// TwinCAT 3 PLC project Samples
// Title: TF8040 PLC-Samples
// Company: Beckhoff Automation GmbH
// Author: Beckhoff Automation
// ProjectVersion: 2.1.2.0
// Description: PLC.Samples to demontrate function volume of TF8040.
// ProgramVersion: 3.1.4026.20
// libraries:
//   Tc2_Standard, * (Beckhoff Automation GmbH)
//   Tc2_System, * (Beckhoff Automation GmbH)
//   Tc2_Utilities, * (Beckhoff Automation GmbH)
//   Tc3_BA2, * (Beckhoff Automation GmbH)
//   Tc3_BA2_Common, * (Beckhoff Automation GmbH)
//   Tc3_BACnetRev14, * (Beckhoff Automation GmbH)
//   Tc3_Module, * (Beckhoff Automation GmbH)
//   Tc3_XBA, * (Beckhoff Automation GmbH)
// project tree:
//   / PlcTask.TcTTO (not stored)
//   SAMPLES/Demo/Event/ FB_Evt_Ack.TcPOU, FB_Evt_EventClasses.TcPOU (not stored), FB_Evt_Events.TcPOU (not stored), FB_Evt_Misc.TcPOU, FB_Evt_QueryCnd.TcPOU
//   SAMPLES/Demo/Event/Function/ F_AcknowledgeEventClass.TcPOU, F_CountEventClassActive.TcPOU
//   SAMPLES/Demo/Objects/ FB_Obj_AddParam.TcPOU (not stored), FB_Obj_General.TcPOU (not stored), FB_Obj_Misc.TcPOU (not stored), FB_Obj_Sequence.TcPOU (not stored), FB_Obj_UserDefined.TcPOU (not stored)
//   SAMPLES/Demo/Objects/Misc/ E_UDef_Mode.TcDUT, FB_UDef_BValEx.TcPOU (not stored), FB_UDef_SpVal.TcPOU (not stored), FB_UDef_SpValEx.TcPOU
//   SAMPLES/Demo/Optional Extensions/Events/ FB_MyLocalObjectEvents.TcPOU, FB_MyProjectEvents.TcPOU
//   SAMPLES/Demo/Optional Extensions/ MAIN_OPTEXT.TcPOU (not stored)
//   SAMPLES/Demo/Other/ FB_Misc.TcPOU (not stored), FB_Texts.TcPOU
//   SAMPLES/Demo/Plant/ FB_Plt_Init1.TcPOU, FB_Plt_Init2.TcPOU, FB_Plt_Init3.TcPOU (not stored)
//   SAMPLES/Demo/Reference/ FB_Ref_Collectors.TcPOU (not stored), FB_Ref_Groups.TcPOU
//   SAMPLES/Demo/Reference/Publish and Subscribe/ FB_Ref_PubSub_Local.TcPOU, FB_Ref_PubSub_Remote.TcPOU (not stored)
//   SAMPLES/Demo/Structure/ FB_Struct_Nested.TcPOU (not stored)
//   SAMPLES/Demo/Supplements/BACnet/ FB_BACnet_EvtInh.TcPOU (not stored), FB_BACnet_ObjPropRef.TcPOU (not stored), FB_BACnet_ObjPropRef_1.TcPOU (not stored), FB_BACnet_RcpList.TcPOU (not stored)
//   SAMPLES/Demo/Supplements/BACnet/Extensions/Events/ FB_BACnet_MyLocalObjectEvents.TcPOU
//   SAMPLES/Demo/Supplements/BACnet/Extensions/ MAIN_OPTEXT_BACnet.TcPOU (not stored)
//   SAMPLES/Demo/[Helper]/FunctionBlocks/Aggregates/ FB_TimerAggregateA.TcPOU (not stored), FB_ProcAggregateB.TcPOU (not stored)
//   SAMPLES/Demo/[Helper]/FunctionBlocks/Nested/ FB_NestedView.TcPOU (not stored), FB_NestedView2.TcPOU (not stored), FB_SubNestedView.TcPOU (not stored), FB_SubSubNestedView.TcPOU (not stored)
//   SAMPLES/ MAIN.TcPOU
//   SAMPLES/Templates/Standard/DUTs/Enumerations/OpMod/ E_OpMod_AC.TcDUT (not stored), E_OpMod_Binary.TcDUT (not stored), E_OpMod_ClsOpn.TcDUT, E_OpMod_Step2.TcDUT
//   SAMPLES/Templates/Standard/GVLs/ MyECIDs.TcGVL, MyLabels.TcGVL (not stored), MyProfiles.TcGVL (not stored)
//   SAMPLES/Templates/Standard/POUs/Trade/General/Building/ FB_BA_Bld01.TcPOU (not stored)
//   SAMPLES/Templates/Standard/POUs/Trade/General/EventClasses/ FB_BA_EC01.TcPOU
//   SAMPLES/Templates/User-defined/Objects/ FB_UDef_Obj.TcPOU
//   SAMPLES/Templates/User-defined/Sample Weather Station/ FB_BA_MyWeatherStation.TcPOU, FB_BA_MyWeatherStationSub.TcPOU, I_BA_MyWeatherStation.TcIO (not stored), ST_BA_MyWeatherData.TcDUT (not stored)
// real-time tasks:
//   TASK PlcTask: cycle T#45ms, priority 20, ADS port 350
//   TASK Device 1 (BACnet IP)_Task_58: cycle T#40ms, priority 58, ADS port 351
//   TASK Gerät 1 (BACnet IP)_QueueTask: cycle T#2ms, priority 8, ADS port 352
// I/O:
//   DEVICE Gerät 1 (BACnet IP), AmsNetId 10.10.1.201.2.1
// variable links:
//   Samples/Samples Instance <-> Device 1 (BACnet IP)
//     PlcTask Inputs/BACnet_Globals.DefaultAdapter.BACnet_AmsNetId <-> Inputs/AmsNetId

// ---- SAMPLES/Demo/Objects/Misc/E_UDef_Mode.TcDUT
{attribute 'qualified_only'}
{attribute 'strict'}

{attribute 'BaParam.Enum.eAdd.DE' := 'Hinzufügen'}
{attribute 'BaParam.Enum.eAdd.EN' := 'Add'}
{attribute 'BaParam.Enum.eSubstract.DE' := 'Abziehen'}
{attribute 'BaParam.Enum.eSubstract.EN' := 'Substract'}
TYPE E_UDef_Mode :
(
	eAdd,
	eSubstract
);
END_TYPE

// ---- SAMPLES/Templates/Standard/DUTs/Enumerations/OpMod/E_OpMod_ClsOpn.TcDUT
{attribute 'qualified_only'}
TYPE E_OpMod_ClsOpn :
(
	eClose			:= 0,
	eOpen			:= 1
	
) UDINT;
END_TYPE

// ---- SAMPLES/Templates/Standard/DUTs/Enumerations/OpMod/E_OpMod_Step2.TcDUT
{attribute 'qualified_only'}
TYPE E_OpMod_Step2 :
(
	Invalid			:= 0,
	
	eOff			:= 1,
	eStep1			:= 2,
	eStep2			:= 3
	
) UDINT;
END_TYPE

// ---- SAMPLES/Templates/Standard/GVLs/MyECIDs.TcGVL
{attribute 'qualified_only'}
VAR_GLOBAL CONSTANT
	AlmSmpl						: UDINT := 112;
	AlmStd						: UDINT := 111;
	AlmExt						: UDINT := 110;
	
	DstSmpl						: UDINT := 122;
	DstStd						: UDINT := 121;	
	DstExt						: UDINT := 120;
	
	MntnSmpl					: UDINT := 132;
	MntnStd						: UDINT := 131;
	MntnExt						: UDINT := 130;
	
	NtfSmpl						: UDINT := 141;
	NtfStd						: UDINT := 140;
	
	OthSmpl						: UDINT := 151;
	OthStd						: UDINT := 150;
END_VAR

// ---- SAMPLES/Demo/Event/FB_Evt_Ack.TcPOU
// Acknowledgement-Examples.
// > One object per demonstrated 'AlarmMode'.
// > See "FB_BA_EC01" to view decleared event classes.
// [Hint]
// > All reference-variables are implemented to ease monitoring of relevant variables.
// > show the possibility to acknowledge BA objects assigned to a specific event class.
FUNCTION_BLOCK FB_Evt_Ack EXTENDS FB_BA_View
VAR               
	{region 'General'}
		bAlm_Test						: BOOL;																						// Trigger alarm for testing.
		bAlm_AckAll						: REFERENCE TO BOOL							REF= THIS^.bAcknowledgeRm;						// Acknowledge all test objects.
		bAlm_AckMode					: POINTER TO BOOL							:= ADR(XBA_Param.eEvtMgmt_AckMode);				// Used reset mode (See parameter description for more details)
	{endregion}
		 
	{region 'Simple'}
		// Intention:					Alarm that automatically disappears.
		// State on active alarm:		- "bEvent = TRUE'
		//								- "stAckedTransitions = [FALSE,true,true]'
		// State when disappeared:		- "bEvent = false'
		//								- "stAckedTransitions = [true,true,true]'
		AlmSimple_Ack					: REFERENCE TO BOOL							REF= AlmSimple.bAcknowledgeRm;
		AlmSimple_Indicated				: BOOL;
		AlmSimple_Event					: REFERENCE TO BOOL							REF= AlmSimple.bEvent;
		AlmSimple						: FB_BA_BI_Raw := (
											iParent									:= THIS^,
											sInactiveText							:= 'Normal',
											sActiveText								:= 'Alarm',
											nEventClassID							:= MyECIDs.AlmSmpl);
	{endregion}
	{region 'Standard'}
		// Intention:					Alarm that is just indicated (by acknowledge transition) when disappeared.
		// State on active alarm:		- "bEvent = TRUE'
		//								- "stAckedTransitions = [FALSE,true,true]'
		// State when disappeared:		- "bEvent = false'
		//								- "stAckedTransitions = [FALSE,true,true]'
		// State after acknowledgement:	- "bEvent = false'
		//								- "stAckedTransitions = [true,true,true]'
		AlmStandard_Ack					: REFERENCE TO BOOL							REF= AlmStandard.bAcknowledgeRm;
		AlmStandard_Indicated			: BOOL;
		AlmStandard_Event				: REFERENCE TO BOOL							REF= AlmStandard.bEvent;
		AlmStandard						: FB_BA_BI_Raw := (
											iParent									:= THIS^,
											sInactiveText							:= 'Normal',
											sActiveText								:= 'Alarm',
											nEventClassID							:= MyECIDs.AlmStd);	
	{endregion}
	{region 'Extended'}
		// Intention:					Alarm that is indicated (by acknowledge transition) and hold when disappeared.
		//								The 'bEvent' is released when an additional reset has been triggered.
		// State on active alarm:		- "bEvent = TRUE'
		//								- "stAckedTransitions = [FALSE,true,FALSE]'
		// State when disappeared:		- "bEvent = TRUE'
		//								- "stAckedTransitions = [FALSE,true,FALSE]'
		// State after acknowledgement:	- "bEvent = TRUE'
		//								- "stAckedTransitions = [true,true,FALSE]'
		// State after reset:			- "bEvent = false'
		//								- "stAckedTransitions = [true,true,true]'
		AlmExtended_Ack					: REFERENCE TO BOOL							REF= AlmExtended.bAcknowledgeRm;
		AlmExtended_Indicated			: BOOL;
		AlmExtended_Event				: REFERENCE TO BOOL							REF= AlmExtended.bEvent;
		AlmExtended						: FB_BA_BI_Raw := (
											iParent									:= THIS^,
											sInactiveText							:= 'Normal',
											sActiveText								:= 'Alarm',
											nEventClassID							:= MyECIDs.AlmExt);	
	{endregion}	
		 
	{region 'Acknowledge event class'}	
		// Intention:					Acknowledge all objects that reference a specific event class.
		nEventClassID					: UINT										:= 0;			// Enter ID of event class to acknowledge.
	{endregion}
	{region 'count active events of event class'}	
		// Intention:					count all objects with active events reference a specific event class.
		nEvents							: UINT;		//count of events of specific class 
	{endregion} 	
END_VAR

SUPER^();

AlmSimple(bRawVal:=bAlm_Test);
AlmSimple_Indicated := (NOT AlmSimple.stAckedTransitions.bToOffnormal);
AlmStandard(bRawVal:=bAlm_Test);
AlmStandard_Indicated := (NOT AlmStandard.stAckedTransitions.bToOffnormal);
AlmExtended(bRawVal:=bAlm_Test);
AlmExtended_Indicated := (NOT AlmExtended.stAckedTransitions.bToOffnormal);

IF (nEventClassID <> 0) THEN
	F_AcknowledgeEventClass(nEventClassID);
	nEventClassID := 0;
END_IF

nEvents:= F_CountEventClassActive(nEventClassID);

// Intention:			Illustrate how to recognize changed events.
METHOD PROTECTED OnObjectEventChange
VAR_INPUT
	iObject				: I_BA_EventObject;
	bNotifyParents		: BOOL				:= TRUE;
END_VAR
SUPER^.OnObjectEventChange(iObject, bNotifyParents);

// Sample 1) Evaluate current event state:
CASE (iObject.EventIcon.eState) OF
	E_BA_EventIconState.eGoneAcked,
	E_BA_EventIconState.ePresentAcked:
		iObject.LogMsg.Show(ADSLOG_MSGTYPE_HINT, 'OOEC06', 'Object acknowledged.', TRUE);
END_CASE

// Sample 2) Compare actual event state to previous event state:
IF (iObject.LastEventIcon.eState < iObject.EventIcon.eState) THEN
	; // State intensed...
ELSE
	; // State softened...
END_IF
END_METHOD

END_FUNCTION_BLOCK

// ---- SAMPLES/Demo/Event/Function/F_AcknowledgeEventClass.TcPOU
// Acknowledge all event class related objects.
FUNCTION F_AcknowledgeEventClass  
VAR_INPUT
	nEventClassID		: UINT					:= 0;		// Target event class ID.
END_VAR
VAR
	_iObj				: I_BA_Object;
	_iEvtObj			: I_BA_EventObject;
END_VAR

// Iterate over all objects:
WHILE (F_BA_IterateObjects(_iObj)) DO
	IF (NOT __QUERYINTERFACE(_iObj,_iEvtObj)) THEN
		;	     
	ELSIF (_iEvtObj.EventClassID <> nEventClassID) THEN
		; // Skip.
	ELSE
		_iEvtObj.AcknowledgeRm := TRUE;
	END_IF
END_WHILE

END_FUNCTION

// ---- SAMPLES/Demo/Event/Function/F_CountEventClassActive.TcPOU
// Count all event class related objects with active events.
FUNCTION F_CountEventClassActive  :UINT
VAR_INPUT
	nEventClassID		: UINT					:= 0;		// Target event class ID.
END_VAR
VAR
	_nEvents			: UINT;
	_iObj				: I_BA_Object;
	_iEvtObj			: I_BA_EventObject;
END_VAR

// Iterate over all objects:
_nEvents := 0;
WHILE (F_BA_IterateObjects(_iObj)) DO
	IF (NOT __QUERYINTERFACE(_iObj,_iEvtObj)) THEN
		; // Skip.	     
	ELSIF (_iEvtObj.EventClassID <> nEventClassID) THEN
		; // Skip.
	ELSIF (_iEvtObj.Event = FALSE) THEN
		; // Skip.
	ELSE
		_nEvents := _nEvents+1;
	END_IF
END_WHILE
F_CountEventClassActive:=_nEvents;

END_FUNCTION

// ---- SAMPLES/Demo/Event/FB_Evt_Misc.TcPOU
FUNCTION_BLOCK FB_Evt_Misc EXTENDS FB_BA_View
VAR
	{region 'Iteration'}
		// Intention:			Iterate over active events.
		bIterate				: BOOL;
		bIterate_ShowTimestamp	: BOOL				:= FALSE;
		bIterate_ShowType		: BOOL				:= TRUE;
		bIterate_ShowState		: BOOL				:= TRUE;
		bIterate_ShowEC			: BOOL				:= FALSE;
	{endregion}
END_VAR
VAR
	_i							: DINT;
	_sVal						: T_MaxString;
	_iObj						: I_BA_EventObject;
	_fbMsg						: FB_BA_DecorString;
END_VAR

SUPER^();

IF (bIterate) THEN
	bIterate := FALSE;
	
	_i := F_BA_GetEventCount();
	IF (_i = 0) THEN
		F_BA_LogMessage(ADSLOG_MSGTYPE_HINT, 'EM06', 'No active events found yet.');
	ELSE
		F_BA_LogMessage1(ADSLOG_MSGTYPE_HINT, 'EM08', 'Active events: %d', F_DINT(_i));
		
		// Iterate over all active events:
		_i := 0;
		_iObj := 0;								// [Hint] Temporary iterator-object must be NULL to start iteration from the beginning.
		WHILE (F_BA_IterateEvents(_iObj)) DO
			_i := (_i+1);
			
			// Format message:
			_fbMsg.Reset();
			IF (bIterate_ShowTimestamp) THEN
				_sVal := TO_STRING(F_BA_ToDT(_iObj.EventChangeTime));
				_fbMsg.AddDecor1('%s', F_STRING(_sVal));
			END_IF
			IF (bIterate_ShowType) THEN
				_fbMsg.AddDecor1('Type: %s', F_STRINGEx(XBA_EnumEN.aEventType[_iObj.EventIcon.eEventType].sName));
			END_IF
			IF (bIterate_ShowState) THEN
				_fbMsg.AddDecor1('State: %s', F_STRINGEx(XBA_EnumEN.aEventIconState[_iObj.EventIcon.eState].sDescription));
			END_IF
			IF (bIterate_ShowEC) THEN
				_sVal := TO_STRING(_iObj.EventClassID);
				_fbMsg.AddDecor1('Event class: %s', F_STRING(_sVal));
			END_IF
			_fbMsg.Finish();
			
			_sVal := _iObj.ObjectName;
			F_BA_LogMessage3(ADSLOG_MSGTYPE_HINT, 'EM32', '%d. %s   %s', F_DINT(_i), F_STRING(_sVal), F_STRING(_fbMsg.sOutput));
		END_WHILE
	END_IF
END_IF

END_FUNCTION_BLOCK

// ---- SAMPLES/Demo/Event/FB_Evt_QueryCnd.TcPOU
// Determine some view's event conditions.
// Intention:
// - Illustrate how to determine (cumulative) event information of a view instance.
FUNCTION_BLOCK FB_Evt_QueryCnd
VAR	
	bUpdate			: BOOL;
	
	{region 'Settings'}
		iSource		: I_BA_View		:= MAIN.Evt;			// Instance to be queried for informations (This can be any view).
	{endregion}
	{region 'Result'}
		nAlarms		: UINT;									// Count of active alarms.
		nOverridden	: UINT;									// Count of overridden objects.
		nCritical	: UINT;									// Count of objects in "Critical" priority.
	{endregion}
END_VAR

IF (bUpdate) AND_THEN (iSource <> 0) THEN
	nAlarms := iSource.EventConditionCount(E_BA_EventCondition.eTypeAlarm);
	nOverridden := iSource.EventConditionCount(E_BA_EventCondition.eFlagOverridden);
	nCritical := iSource.EventConditionCount(E_BA_EventCondition.ePrioCritical);
END_IF

bUpdate := FALSE;

END_FUNCTION_BLOCK

// ---- SAMPLES/MAIN.TcPOU
PROGRAM MAIN
VAR
	{region 'Settings'}
		DPAD						: FB_BA_CarelessDPAD:=(
										aIdentifier:=[
											(* Level 1 *)	(eNodeType:=E_BA_NodeType.eBuilding,	nIndexDigits:=2),
											(* Level 2 *)	(eNodeType:=E_BA_NodeType.eTrade,		nIndexDigits:=0),
											(* Level 3 *)	(eNodeType:=E_BA_NodeType.ePlant,		nIndexDigits:=2,			sSeparator_ObjectName:='~~~',		sSeparator_Description:=' --- '),
											(* Level 4 *)	(eNodeType:=E_BA_NodeType.eAggregate,	nIndexDigits:=2,			sSeparator_ObjectName:='++'),
											(* Level 5 *)	(eNodeType:=E_BA_NodeType.eFunction,	nIndexDigits:=3)
									]);
	{endregion}
		 
	Smpl							: FB_BA_View			:= (									sDescription:='Samples');
	{region 'Demonstration'}
		Demo						: FB_BA_View			:= (iParent:=Smpl,						sDescription:='Demonstration');
			Obj						: FB_BA_View			:= (iParent:=Demo,						sDescription:='Objects');
				General				: FB_Obj_General		:= (iParent:=Obj,						sDescription:='General objects');
				Misc				: FB_Obj_Misc			:= (iParent:=Obj,						sDescription:='Miscellaneous objects');
				Seq					: FB_Obj_Sequence		:= (iParent:=Obj,						sDescription:='Sequences');
				UdObj				: FB_Obj_UserDefined	:= (iParent:=Obj,						sDescription:='User defined objects');
				AddParam			: FB_Obj_AddParam		:= (iParent:=Obj,						sDescription:='Additional parameters');

			Ref						: FB_BA_View			:= (iParent:=Demo,						sDescription:='Reference');
				Collect				: FB_Ref_Collectors		:= (iParent:=Ref,						sDescription:='Collectors');
				Groups				: FB_Ref_Groups			:= (iParent:=Ref,						sDescription:='Groups');
				PubSubLc			: FB_Ref_PubSub_Local	:= (iParent:=Ref,						sDescription:='Publisher and subscriber (Local)');
				PubSubRm			: FB_Ref_PubSub_Remote	:= (iParent:=Ref,						sDescription:='Publisher and subscriber (Remote)');

			Evt						: FB_BA_View			:= (iParent:=Demo,						sDescription:='Event');
				EvtCls				: FB_Evt_EventClasses	:= (iParent:=Evt,						sDescription:='Event classes');
				Events				: FB_Evt_Events			:= (iParent:=Evt,						sDescription:='Events');
				Ack					: FB_Evt_Ack			:= (iParent:=Evt,						sDescription:='Acknowledgement');
				MiscEvt				: FB_Evt_Misc			:= (iParent:=Evt,						sDescription:='Miscellaneous');
				Cnd					: FB_Evt_QueryCnd;

			Strct					: FB_BA_View			:= (iParent:=Demo,						sDescription:='Structure');
				Nested				: FB_Struct_Nested		:= (iParent:=Strct,						sDescription:='Nested objects');

			Plt						: FB_BA_View			:= (iParent:=Demo,						sDescription:='Plant');
				//PltCtrl1			: FB_Plt_Init1			:= (iParent:=Plt,						sDescription:='Plant control initialization 1');
				PltCtrl2			: FB_Plt_Init2			:= (iParent:=Plt,						sDescription:='Plant control initialization 2');
				//PltCtrl3			: FB_Plt_Init3			:= (iParent:=Plt,						sDescription:='Plant control initialization 3');

			Spl						: FB_BA_View			:= (iParent:=Demo,						sDescription:='Supplement specific');
				BACnet_RcpList		: FB_BACnet_RcpList		:= (iParent:=Spl,						sDescription:='Write Recipient list (BACnet)');
				BACnet_ObjPropRef	: FB_BACnet_ObjPropRef	:= (iParent:=Spl,						sDescription:='Write object property reference (BACnet)');
				BACnet_EvtInh		: FB_BACnet_EvtInh		:= (iParent:=Spl,						sDescription:='Write EventInhibit property (BACnet)');
					 
			Other					: FB_BA_View			:= (iParent:=Demo,						sDescription:='Other');
				Texts				: FB_Texts				:= (iParent:=Other,						sDescription:='Name and description texts');
				MscOth				: FB_Misc				:= (iParent:=Other,						sDescription:='Miscellaneous');
	{endregion}
	{region 'Templates'}
		Tmpl						: FB_BA_View			:= (iParent:=Smpl,						sDescription:='Templates');
			Gen						: FB_BA_View			:= (iParent:=Tmpl,						sDescription:='General');
				Bld01				: FB_BA_Bld01			:= (iParent:=Gen,						sDescription:='Building information');
				EvtCls01			: FB_BA_EC01			:= (iParent:=Gen,						sDescription:='Event Classes');
	{endregion}		
END_VAR
VAR		
	nCounter						: UDINT					:= 0;	
END_VAR

nCounter:=(nCounter+1);

Smpl();

// Demonstration:
Demo();

Obj();
General();
Misc();
Seq();
UdObj();
AddParam();

Ref();
Collect();
Groups();
PubSubLc();
PubSubRm();

Evt();
EvtCls();
Events();
Ack();
MiscEvt();
Cnd();

Strct();
Nested();

Plt();
//PltCtrl1();
PltCtrl2();
//PltCtrl3();

Spl();
BACnet_RcpList();
BACnet_ObjPropRef();
BACnet_EvtInh();

Other();
Texts();
MscOth();

// Templates:
Tmpl();

Gen();
Bld01();
EvtCls01();

// Optional extensions:
MAIN_OPTEXT();
MAIN_OPTEXT_BACnet();

END_PROGRAM

// ---- SAMPLES/Demo/Reference/FB_Ref_Groups.TcPOU
// Examples of groups.
FUNCTION_BLOCK FB_Ref_Groups EXTENDS FB_BA_View
VAR
	{region 'Analog'}
		A							: FB_BA_View := (
										iParent							:= THIS^,
										sDescription					:= '{Analog objects}'
									);
				                    
			GrpAV1					: FB_BA_AV := (
										iParent							:= A,
										eUnit							:= E_BA_Unit.eOther_NoUnits,
										nEventClassID					:= MyECIDs.AlmStd,
										bEnPgm							:= TRUE,
										fValPgm							:= 10
									);
			GrpAV2					: FB_BA_AV := (
										iParent							:= A,
										eUnit							:= E_BA_Unit.eOther_NoUnits,
										nEventClassID					:= MyECIDs.AlmStd,
										bEnPgm							:= TRUE,
										fValPgm							:= 15
									);
			GrpAVOp1				: FB_BA_AV_Op := (
										iParent							:= A,
										eUnit							:= E_BA_Unit.eTemperature_DegreesCelsius,
										fValueRm						:= 20
									);
			GrpAVOp2				: FB_BA_AV_Op := (
										iParent							:= A,
										eUnit							:= E_BA_Unit.eTemperature_DegreesCelsius,
										fValueRm						:= 25
									);
										 
			// Intention:			Eigenständige Gruppe (Ohne Achsen-Zugehörigkeit)
			Group_AVMin				: FB_BA_Group_AVal := (
										eCalcMode						:= E_BA_AValCalcMode.eMin,
										iReference						:= [ GrpAV1, GrpAV2, GrpAVOp1, GrpAVOp2 ]
									);
			Group_AVMax				: FB_BA_Group_AVal := (
										eCalcMode						:= E_BA_AValCalcMode.eMax,
										iReference						:= [ GrpAV1, GrpAV2, GrpAVOp1, GrpAVOp2 ]
									);
			Group_AVAvg				: FB_BA_Group_AVal := (
										eCalcMode						:= E_BA_AValCalcMode.eAverage,
										iReference						:= [ GrpAV1, GrpAV2, GrpAVOp1, GrpAVOp2 ]
									);
	{endregion}
END_VAR

SUPER^(); // FB_BA_View
A(); // FB_BA_View
GrpAV1(); // FB_BA_AV
GrpAV2(); // FB_BA_AV
GrpAVOp1(); // FB_BA_AV_Op
GrpAVOp2(); // FB_BA_AV_Op
Group_AVMin(); // FB_BA_Group_AVal
Group_AVMax(); // FB_BA_Group_AVal
Group_AVAvg(); // FB_BA_Group_AVal

END_FUNCTION_BLOCK

// ---- SAMPLES/Demo/Reference/Publish and Subscribe/FB_Ref_PubSub_Local.TcPOU
// Example of internal device communication.
FUNCTION_BLOCK FB_Ref_PubSub_Local EXTENDS FB_BA_View
VAR
	{region 'Analog'}
	
		A								: FB_BA_View := (
											iParent						:= THIS^,
											sDescription				:= '{Analog objects}'
										);
													 
			AV_Sub						: FB_BA_SubAPrio				:= (sSubject:='AV_Obj');
			AV_Obj						: FB_BA_AV := (
											iParent						:= A,
											iProfile					:= MyProfiles.AV_Prf,
											bEnPublish					:= TRUE
										); 
			AVOp_Sub					: FB_BA_SubAV_Op				:= (sSubject:='AVOp_Obj');
			AVOp_Obj					: FB_BA_AV_Op := (
											iParent						:= A,
											iProfile					:= MyProfiles.AVOp_Prf,
											bEnPublish					:= TRUE,
											fValueRm					:= 10
										); 
			AI_Sub						: FB_BA_SubAI					:= (sSubject:='AI_Obj');
			AI_Obj						: FB_BA_AI_Raw := (
											iParent						:= A,
											iProfile					:= MyProfiles.AI_Prf,
											bEnPublish					:= TRUE
										); 
			AO_Sub						: FB_BA_SubAPrio				:= (sSubject:='AO_Obj');
			AO_Obj						: FB_BA_AO_Raw := (
											iParent						:= A,
											iProfile					:= MyProfiles.AO_Prf,
											bEnPublish					:= TRUE
										); 
	{endregion}
	{region 'Binary'}
		B								: FB_BA_View := (
											iParent						:= THIS^,
											sDescription				:= '{Binary objects}'
										);
												 
			BV_Sub						: FB_BA_SubBPrio				:= (sSubject:='BV_Obj'); 
			BV_Obj						: FB_BA_BV := (
											iParent						:= B,
											iProfile					:= MyProfiles.BV_Prf,
											bEnPublish					:= TRUE
										);
			BVOp_Sub					: FB_BA_SubBV_Op				:= (sSubject:='BVOp_Obj');
			BVOp_Obj					: FB_BA_BV_Op := (
											iParent						:= B,
											iProfile					:= MyProfiles.BVOp_Prf,
											bEnPublish					:= TRUE,
											bValueRm					:= TRUE
										);
			BI_Sub						: FB_BA_SubBI					:= (sSubject:='BI_Obj');
			BI_Obj						: FB_BA_BI_Raw := (
											iParent						:= B,
											iProfile					:= MyProfiles.BI_Prf,
											bEnPublish					:= TRUE
										);
			BO_Sub						: FB_BA_SubBPrio				:= (sSubject:='BO_Obj');
			BO_Obj						: FB_BA_BO_Raw := (
											iParent						:= B,
											iProfile					:= MyProfiles.BO_Prf,
											bEnPublish					:= TRUE
										); 
	{endregion}
	{region 'Multistate'}
		M								: FB_BA_View := (
											iParent						:= THIS^,
											sDescription				:= '{Multistate objects}'
										);
			 
			MV_Sub						: FB_BA_SubMPrio				:= (sSubject:='MV_Obj');
			MV_Obj						: FB_BA_MV := (
											iParent						:= M,
											iProfile					:= MyProfiles.MV_Prf,
											bEnPublish					:= TRUE
										);
			MVOp_Sub					: FB_BA_SubMV_Op				:= (sSubject:='MVOp_Obj');
			MVOp_Obj					: FB_BA_MV_Op := (
											iParent						:= M,
											iProfile					:= MyProfiles.MVOp_Prf,
											bEnPublish					:= TRUE,
											nValueRm					:= 2
										);
			MI_Sub						: FB_BA_SubMI					:= (sSubject:='MI_Obj');
			MI_Obj						: FB_BA_MI_Raw := (
											iParent						:= M,
											iProfile					:= MyProfiles.MI_Prf,
											bEnPublish					:= TRUE
										);
			MO_Sub						: FB_BA_SubMPrio				:= (sSubject:='MO_Obj');
			MO_Obj						: FB_BA_MO_Raw := (
											iParent						:= M,
											iProfile					:= MyProfiles.MO_Prf,
											bEnPublish					:= TRUE
										); 
	{endregion}
	{region 'Miscellaneous'}
		Misc							: FB_BA_View := (
											iParent						:= THIS^,
											sDescription				:= '{Miscellaneous objects}'
										);
			 
			Loop_Sub					: FB_BA_SubLoop					:= (sSubject:='Loop_Obj');
			Loop_Obj					: FB_BA_LoopSeq := (
											iParent						:= Misc,
											iProfile					:= MyProfiles.Loop_Prf,
											bEnPublish					:= TRUE,
											fProportionalConstant		:= 5.0,
											fIntegralConstant			:= 180,
											bEn							:= TRUE,
											fSetpoint					:= 20,
											fCtrlVal					:= 25
										);
	                                    
			Cal_Sub						: FB_BA_SubCal					:= (sSubject:='Cal_Obj');
			Cal_Obj						: FB_BA_Cal := (
											iParent						:= Misc,
											iProfile					:= MyProfiles.Cal_Prf,
											bEnPublish					:= TRUE,
											aDateList := [(
												eType					:= E_BA_DateValChoice.eWeekNDay,
												uDate					:= F_BA_WeekNDayVal(E_BA_Weekday.eFriday, E_BA_Week.eWeek1, E_BA_Month.eFebruary)
											)]);
												 
			SchedA_Sub					: FB_BA_SubSchedA				:= (sSubject:='SchedA_Obj');
			SchedA_Obj					: FB_BA_SchedA := (
											iParent						:= Misc,
											iProfile					:= MyProfiles.SchedA_Prf,
											bEnPublish					:= TRUE,
											aWeek						:= F_BA_SchedWeekly3xA(E_BA_Weekday.eMonday, E_BA_Weekday.eFriday, T#0H, 0.0, T#6H, 5.0, T#20H, 0.0));
			SchedB_Sub					: FB_BA_SubSchedB				:= (sSubject:='SchedB_Obj');
			SchedB_Obj					: FB_BA_SchedB := (
											iParent						:= Misc,
											iProfile					:= MyProfiles.SchedB_Prf,
											bEnPublish					:= TRUE,
											aWeek						:= F_BA_SchedWeekly3xB(E_BA_Weekday.eMonday, E_BA_Weekday.eFriday, T#0H, FALSE, T#6H, TRUE, T#20H, FALSE));
			SchedM_Sub					: FB_BA_SubSchedM				:= (sSubject:='SchedM_Obj');
			SchedM_Obj					: FB_BA_SchedM := (
											iParent						:= Misc,
											iProfile					:= MyProfiles.SchedM_Prf,
											bEnPublish					:= TRUE,
											aWeek						:= F_BA_SchedWeekly3xM(E_BA_Weekday.eMonday, E_BA_Weekday.eFriday, T#0H, 1, T#6H, 2, T#20H, 1));
												 
			Trend_Sub					: FB_BA_SubTrend				:= (sSubject:='Trend_Obj');
			Trend_Obj					: FB_BA_Trend := (
											iParent						:= Misc,
											iProfile					:= MyProfiles.Trend_Prf,
											bEnPublish					:= TRUE,
											nEventClassID				:= MyECIDs.AlmStd,
											stReferencedParam			:= F_BA_Reference(AV_Obj, E_BA_Parameter.ePresentValue)
										);
	{endregion}
	{region 'Custom'}
		{region 'Typed'}
			MyWthSt						: FB_BA_MyWeatherStation		:= (bEnPublish:= TRUE); 
			MyWthSt_Sub					: FB_BA_MyWeatherStationSub		:= (sSubject:='MyWthSt');
		{endregion}
		{region 'Raw'}
			MyRawWthStData				: ST_BA_MyWeatherData;
			MyRawWthSt					: FB_BA_RawPublisher;
					  
			MyRawWthStData_Sub			: ST_BA_MyWeatherData;
			MyRawWthSt_Sub				: FB_BA_RawSubscriber			:= (sSubject:='MyRawWthSt');
		{endregion}
	{endregion}
	{region 'Tests'}
		Tests							: FB_BA_View := (
											iParent						:= THIS^,
											sDescription				:= '{Test objects}'
										);
			 
		{region 'Subject path'}
			Nested1a					: FB_NestedView := (
											View						:= (iParent := Tests),
											Value						:= (bEnPublish := TRUE)
										);
			Nested1b					: FB_NestedView := (
											View						:= (iParent := Tests),
											Value						:= (bEnPublish := TRUE)
										);

			Nested1a_AV_Sub				: FB_BA_SubAV_Op := (
										//	sSubject					:= 'Value'							// -> Would lead to ambiguous subject!
											sSubject					:= 'Nested1a.Value'
										);
		{endregion}
	{endregion}
END_VAR

SUPER^(); // FB_BA_View
A(); // FB_BA_View
AO_Obj(); // FB_BA_AO_Raw
AV_Obj(); // FB_BA_AV
AI_Obj(); // FB_BA_AI_Raw
AVOp_Obj(); // FB_BA_AV_Op
AO_Sub(); // FB_BA_SubAPrio
AV_Sub(); // FB_BA_SubAPrio
AVOp_Sub(); // FB_BA_SubAV_Op
AI_Sub(); // FB_BA_SubAI
B(); // FB_BA_View
BO_Obj(); // FB_BA_BO_Raw
BV_Obj(); // FB_BA_BV
BI_Obj(); // FB_BA_BI_Raw
BVOp_Obj(); // FB_BA_BV_Op
BO_Sub(); // FB_BA_SubBPrio
BV_Sub(); // FB_BA_SubBPrio
BVOp_Sub(); // FB_BA_SubBV_Op
BI_Sub(); // FB_BA_SubBI
M(); // FB_BA_View
MO_Obj(); // FB_BA_MO_Raw
MV_Obj(); // FB_BA_MV
MI_Obj(); // FB_BA_MI_Raw
MVOp_Obj(); // FB_BA_MV_Op
MO_Sub(); // FB_BA_SubMPrio
MV_Sub(); // FB_BA_SubMPrio
MVOp_Sub(); // FB_BA_SubMV_Op
MI_Sub(); // FB_BA_SubMI
Misc(); // FB_BA_View
Loop_Obj(); // FB_BA_LoopSeq
Trend_Obj(); // FB_BA_Trend
SchedA_Obj(); // FB_BA_SchedA
SchedB_Obj(); // FB_BA_SchedB
SchedM_Obj(); // FB_BA_SchedM
Cal_Obj(); // FB_BA_Cal
Loop_Sub(); // FB_BA_SubLoop
Cal_Sub(); // FB_BA_SubCal
SchedA_Sub(); // FB_BA_SubSchedA
SchedB_Sub(); // FB_BA_SubSchedB
SchedM_Sub(); // FB_BA_SubSchedM
Trend_Sub(); // FB_BA_SubTrend
MyWthSt(); // FB_BA_MyWeatherStation
// Copy some weather data to get nice (=simulated) values - just for this demo.
MyRawWthStData := MyWthSt.stData;
MyRawWthSt(xData := MyRawWthStData); // FB_BA_RawPublisher
MyRawWthSt_Sub(xData := MyRawWthStData_Sub); // FB_BA_RawSubscriber
MyWthSt_Sub(); // FB_BA_MyWeatherStationSub
Tests(); // FB_BA_View
Nested1a(); // FB_NestedView
Nested1a_AV_Sub(); // FB_BA_SubAV_Op
Nested1b(); // FB_NestedView

END_FUNCTION_BLOCK

// ---- SAMPLES/Templates/User-defined/Sample Weather Station/FB_BA_MyWeatherStation.TcPOU
// [Sample]
// User specific weather station.
FUNCTION_BLOCK FB_BA_MyWeatherStation EXTENDS FB_BA_Publisher IMPLEMENTS I_BA_MyWeatherStation
VAR_OUTPUT
	fWeatherTemperature	: REAL;
	fHumidity			: REAL;
	fBrightness			: REAL;
	
	bDisturb			: BOOL;
END_VAR
VAR
	{region 'Internal'}
		eState			: (eInit:=1, eOperation:=2, eError:=3) UDINT	:= 1;
		stData			: ST_BA_MyWeatherData;
	{endregion}
	{region 'Temporary'}
		_nCounter		: UINT;
	{endregion}
END_VAR

CASE (eState) OF
	eInit:
		IF (OnInit()) THEN
			eState := eOperation;
		ELSE
			eState := eError;
		END_IF
		
	eOperation:
		// [Sample] Simulate weather data.
		_nCounter := (_nCounter+1);
		
		IF ((_nCounter MOD 1000) > 800) THEN
			// Simulate a physical error:
			MEMSET(ADR(stData), 0, SIZEOF(stData));
			stData.fWeatherTemperature := 99.9;
			stData.fHumidity := 99.9;
			stData.bDisturb := TRUE;
		ELSE
			// Simulate valid values:
			stData.fWeatherTemperature := 20 + (TO_REAL((_nCounter / 10) MOD 100) * 0.01);
			stData.fHumidity := TO_REAL(50 + (_nCounter MOD 1000) / 500);
			stData.fBrightness := TO_REAL(10 + (_nCounter MOD 1000) / 200);
			stData.fWindSpeed := TO_REAL(5 + ((_nCounter MOD 500) / 10));
			stData.fWindDirection := TO_REAL(90 + ((_nCounter MOD 500) / 200));
			stData.fLatitude := 51.8761551;
			stData.fLongitude := 8.4671055;
			stData.bDisturb := FALSE;
		END_IF
		
END_CASE
		
// Update outputs of most important variables:
fWeatherTemperature := stData.fWeatherTemperature;
fHumidity := stData.fHumidity;
fBrightness := stData.fBrightness;
bDisturb := stData.bDisturb;

PROPERTY Brightness : REAL
GET
Brightness := stData.fBrightness;
END_GET
END_PROPERTY

PROPERTY Error : BOOL
GET
Error := (eState=eError);
END_GET
END_PROPERTY

METHOD FB_init : BOOL
VAR_INPUT
	bInitRetains : BOOL; // if TRUE, the retain variables are initialized (warm start / cold start)
	bInCopyCode : BOOL;  // if TRUE, the instance afterwards gets moved into the copy code (online change)
END_VAR
// [Hint]
// > Eigentlich wird an dieser Stelle das Profil definiert. Aber zur Übersicht wird es in "MAIN_SharedInterfaces" initialisiert.

// bEnPublish := TRUE;
// iProfile := SampleMyProfiles.MyWeatherStation;
END_METHOD

// Returns published data.
METHOD GetData
VAR_OUTPUT
	pData			: PVOID;				// Pointer to published data.
	nSize			: DINT;					// Size of published data.
END_VAR
pData := ADR(stData);
nSize := SIZEOF(stData);
END_METHOD

PROPERTY Humidity : REAL
GET
Humidity := stData.fHumidity;
END_GET
END_PROPERTY

PROPERTY Latitude : REAL
GET
Latitude := stData.fLatitude;
END_GET
END_PROPERTY

PROPERTY Longitude : REAL
GET
Longitude := stData.fLongitude;
END_GET
END_PROPERTY

METHOD PROTECTED OnInit : BOOL
IF (SUPER^.OnInit()) THEN
	// [Sample]:
	// Implement custom init code here (Optional).
	// ...
	
	OnInit := TRUE;
END_IF
END_METHOD

{attribute 'call_after_online_change_slot' := '5000'}
METHOD PROTECTED OnPostOnlineChange
SUPER^.OnPostOnlineChange();

// Re-initialize after online-changes:
eState := eInit;
END_METHOD

PROPERTY Ready : BOOL
GET
Ready := (eState=eOperation);
END_GET
END_PROPERTY

PROPERTY Valid : BOOL
GET
IF (SUPER^.Valid) THEN
	// [Sample]:
	// Implement custom validation code here (Optional).
	// ...
	
	Valid := TRUE;
END_IF
END_GET
END_PROPERTY

PROPERTY WeatherTemperature : REAL
GET
WeatherTemperature := stData.fWeatherTemperature;
END_GET
END_PROPERTY

PROPERTY WindDirection : REAL
GET
WindDirection := stData.fWindDirection;
END_GET
END_PROPERTY

PROPERTY WindSpeed : REAL
GET
WindSpeed := stData.fWindSpeed;
END_GET
END_PROPERTY

END_FUNCTION_BLOCK

// ---- SAMPLES/Templates/User-defined/Sample Weather Station/FB_BA_MyWeatherStationSub.TcPOU
// [Sample]
// Subscriber to a user specific weather station.
FUNCTION_BLOCK FB_BA_MyWeatherStationSub EXTENDS FB_BA_Subscriber
VAR_OUTPUT
	fWeatherTemperature	: REAL;
	fHumidity			: REAL;
	fBrightness			: REAL;
	
	bDisturb			: BOOL;
END_VAR
VAR
	{region 'General'}
		stData			: ST_BA_MyWeatherData;
	{endregion}
END_VAR

SUPER^();

// Update outputs of most important variables:
fWeatherTemperature := stData.fWeatherTemperature;
fHumidity := stData.fHumidity;
fBrightness := stData.fBrightness;

// Indicate:
// - A physical error that is really occured in the remote weather station
// - A reference error (E.g. broken ADS connection)
bDisturb := (stData.bDisturb) OR (Error);

METHOD FB_init : BOOL
VAR_INPUT
	bInitRetains : BOOL; // if TRUE, the retain variables are initialized (warm start / cold start)
	bInCopyCode : BOOL;  // if TRUE, the instance afterwards gets moved into the copy code (online change)
END_VAR
// [Hint]
// > Eigentlich wird an dieser Stelle das Profil definiert. Aber zur Übersicht wird es in "MAIN_SharedInterfaces" initialisiert.

// iProfile := SampleMyProfiles.MyWeatherStation;
END_METHOD

// Returns subscription-data (For storing read data).
METHOD GetData
VAR_OUTPUT
	pData			: PVOID;				// Pointer to subscribed data.
	nSize			: DINT;					// Size of subscribed data.
END_VAR
pData := ADR(stData);
nSize := SIZEOF(stData);
END_METHOD

METHOD PROTECTED OnValidateSubscription : BOOL
VAR_INPUT
	iPublisher			: I_BA_Publisher;
END_VAR
VAR
	_iSubWthSt			: I_BA_MyWeatherStation;
END_VAR
// Cast interface pointer (Used for a local subscription):
OnValidateSubscription := __QUERYINTERFACE(iPublisher, _iSubWthSt);
END_METHOD

END_FUNCTION_BLOCK

// ---- SAMPLES/Demo/Plant/FB_Plt_Init2.TcPOU
// How to initialize plant control at declaration (Recommended workflow).
// [Hint]
// > All reference-variables are implemented to ease monitoring of relevant variables.
FUNCTION_BLOCK FB_Plt_Init2 EXTENDS FB_BA_View
VAR
   	{region 'Aggregates'}
		DmprSu_Open							: REFERENCE TO BOOL							REF= DmprSu.bOpen;
		DmprSu_Val							: REFERENCE TO REAL							REF= DmprSu.fActiveVal;
		DmprSu								: FB_TimerAggregateA						:= (iParent:=THIS^,					iLabel:=MyLabels.DmprSu);
		FanSu_Val							: REFERENCE TO UDINT						REF= FanSu.nActiveVal;
		FanSu								: FB_BA_AggregateM							:= (iParent:=THIS^,					iLabel:=MyLabels.FanSu);
			 
		DmprEx_Open							: REFERENCE TO BOOL							REF= DmprEx.bOpen;
		DmprEx_Val							: REFERENCE TO REAL							REF= DmprEx.fActiveVal;
		DmprEx								: FB_TimerAggregateA						:= (iParent:=THIS^,					iLabel:=MyLabels.DmprEx);
		FanEx_Val							: REFERENCE TO UDINT						REF= FanEx.nActiveVal;
		FanEx								: FB_BA_AggregateM							:= (iParent:=THIS^,					iLabel:=MyLabels.FanEx);
			 
		PreHtr_Proc							: REFERENCE TO BOOL							REF= PreHtr.Process.bActive;
		PreHtr_Val							: REFERENCE TO BOOL							REF= PreHtr.bActiveVal;
		PreHtr								: FB_ProcAggregateB							:= (iParent:=THIS^,					iLabel:=MyLabels.PreHtr,			Process:=(iLabel:=MyLabels.ProcPreRinse));
		Erc_Val								: REFERENCE TO BOOL							REF= Erc.bActiveVal;
		Erc									: FB_BA_AggregateB							:= (iParent:=THIS^,					iLabel:=MyLabels.Erc);
		Col_Val								: REFERENCE TO BOOL							REF= Col.bActiveVal;
		Col									: FB_BA_AggregateB							:= (iParent:=THIS^,					iLabel:=MyLabels.Col);
	{endregion}
	{region 'Plant'} 
		OpMode								: E_OpMod_AC								:= E_OpMod_AC.eOff;
		PlantCtrl_OpSta						: REFERENCE TO BOOL							REF= PlantCtrl.bOpSta;
		PlantCtrl_On						: REFERENCE TO BOOL							REF= PlantCtrl.bOn;
		PlantCtrl_PrVal						: REFERENCE TO UDINT						REF= PlantCtrl.nPresentValue;
		PlantCtrl_Step						: REFERENCE TO STRING						REF= PlantCtrl.sStep;
		PlantCtrl							: FB_BA_PlantCtrl := (
												iParent									:= THIS^,
												iLabel									:= MyLabels.PltCtrl,
												stOperation := (
													aOpMode								:= [ E_OpMod_AC.eDisturb,				E_OpMod_AC.eSmokeExtract,		E_OpMod_AC.eOff,			E_OpMod_AC.eOn,				E_OpMod_AC.eNightCool ],
													aPriority							:= [ E_BA_Priority.eCritical,			E_BA_Priority.eLifeSafety,		E_BA_Priority.eProgram,		E_BA_Priority.eProgram,		E_BA_Priority.eProgram ],
													aIgnoreFlags						:= [ E_BA_AggregateIgnoreFlags.Delay,	E_BA_AggregateIgnoreFlags.All,	0,							0,							0 ],
													aAggregates := [(
														iReference						:= DmprSu,
														aAggMode						:= [ 0,									100,							0,							100,						100 ]
													), (
														iReference						:= DmprEx,
														aAggMode						:= [ 0,									100,							0,							100,						100 ]
													), (
														iReference						:= PreHtr,
														aAggMode						:= [ E_OpMod_Binary.eOff,				E_OpMod_Binary.eOn,				E_OpMod_Binary.eOff,		E_OpMod_Binary.eOn,			E_OpMod_Binary.eOff ],
														bWaitForProcesses				:= TRUE
													), (
														iReference						:= Erc,
														aAggMode						:= [ E_OpMod_Binary.eOff,				E_OpMod_Binary.eOn,				E_OpMod_Binary.eOff,		E_OpMod_Binary.eOn,			E_OpMod_Binary.eOff ]
													), (
														iReference						:= Col,
														aAggMode						:= [ E_OpMod_Binary.eOff,				E_OpMod_Binary.eOn,				E_OpMod_Binary.eOff,		E_OpMod_Binary.eOn,			E_OpMod_Binary.eOff ]
													), (
														iReference						:= FanSu,
														aAggMode						:= [ E_OpMod_Step2.eOff,				E_OpMod_Step2.eStep2,			E_OpMod_Step2.eOff,			E_OpMod_Step2.eStep1,		E_OpMod_Step2.eStep2 ],
														tDelayStepDown					:= T#0S,
														tDelayStepUp					:= T#5S
													), (
														iReference						:= FanEx,
														aAggMode						:= [ E_OpMod_Step2.eOff,				E_OpMod_Step2.eStep2,			E_OpMod_Step2.eOff,			E_OpMod_Step2.eStep1,		E_OpMod_Step2.eStep2 ],
														tDelayStepDown					:= T#5S,
														tDelayStepUp					:= T#0S
													)]
											));
	{endregion}
END_VAR

SUPER^(); // FB_BA_View
DmprSu(); // FB_TimerAggregateA
FanSu(bEnCrit := NOT DmprSu.bOpen, nValCrit := E_OpMod_Step2.eOff); // FB_BA_AggregateM
DmprEx(); // FB_TimerAggregateA
FanEx(bEnCrit := NOT DmprEx.bOpen, nValCrit := E_OpMod_Step2.eOff); // FB_BA_AggregateM
PreHtr(); // FB_ProcAggregateB
Erc(); // FB_BA_AggregateB
Col(); // FB_BA_AggregateB
PlantCtrl(nOpMode := OpMode); // FB_BA_PlantCtrl

END_FUNCTION_BLOCK

// ---- SAMPLES/Demo/Other/FB_Texts.TcPOU
// Demonstration of concatenating texts like objectname and description.
FUNCTION_BLOCK FB_Texts EXTENDS FB_BA_View
VAR
	{region 'Labels'}
		LblAggregate	: FB_BA_Label			:= (sObjName:='AGG', sDescr:='Aggregate description');
		LblObject		: FB_BA_Label			:= (sObjName:='OBJ', sDescr:='Object description');
	{endregion}
	{region 'Objects'}
		// Intention:	Auto indexing
		//				Default initialization with auto-indexing using labels to get textual information into objectname and description.
		Agg1			: FB_BA_View := (
							iParent				:= THIS^,
							iLabel				:= LblAggregate
						);
			Agg1Obj1	: FB_BA_BV_OP := (
							iParent				:= Agg1,
							iLabel				:= LblObject,
							sInactiveText		:= 'Inaktiv',
							sActiveText			:= 'Aktiv'
						);
			Agg1Obj2	: FB_BA_BV_OP := (
							iParent				:= Agg1,
							iLabel				:= LblObject,
							sInactiveText		:= 'Inaktiv',
							sActiveText			:= 'Aktiv'
						);

		// Intention:	Transfer index information into description using the 'index' attribute.
		Agg2			: FB_BA_View 	:= (
							iParent				:= THIS^,
							iLabel				:= LblAggregate,
							sDescription		:= '{{Idx}}'
						);
			Agg2Obj1	: FB_BA_BV_OP := (
							iParent				:= Agg2,
							iLabel				:= LblObject,
							sDescription		:= '{{Idx}}',
							sInactiveText		:= 'Close',
							sActiveText			:= 'Open'
						);
			Agg2Obj2	: FB_BA_BV_OP := (
							iParent				:= Agg2,
							iLabel				:= LblObject,
							sDescription		:= '{{Idx}}',
							sInactiveText		:= 'Close',
							sActiveText			:= 'Open'
						);

		// Intention:	Set objectname and description without labels but auto-indexing.
		Agg3			: FB_BA_View := (
							iParent				:= THIS^,
							sObjectName	 		:= '{PUM}',
							sDescription		:= '{Pump}'
						);
			Agg3Obj1	: FB_BA_BV_OP := (
							iParent				:= Agg3,
							sObjectName	 		:= '{DST}',
							sDescription		:= '{Disturbance}',
							sInactiveText		:= 'Normal',
							sActiveText			:= 'Disturbance'
						);
			Agg3Obj2	: FB_BA_BV_OP := (
							iParent				:= Agg3,
							sObjectName	 		:= '{OPM}',
							sDescription		:= '{Operation message}',
							sInactiveText		:= 'Off',
							sActiveText			:= 'On'
						);

		// Intention:	Set objectname and description without use of labels and auto-indexing but 'index' attribute.
		Agg4			: FB_BA_View := (
							iParent				:= THIS^,
							sObjectName	 		:= '{PUM{Idx=10}}',
							sDescription		:= '{Pump}'
						);
			Agg4Obj1	: FB_BA_BV_OP := (
							iParent				:= Agg4,
							sObjectName	 		:= '{DST{Idx=10}}',
							sDescription		:= '{Disturbance}',
							sInactiveText		:= 'Normal',
							sActiveText			:= 'Disturbance'
						);
			Agg4Obj2	: FB_BA_BV_OP := (
							iParent				:= Agg4,
							sObjectName	 		:= '{OPM{Idx=20}}',
							sDescription		:= '{Operation message}',
							sInactiveText		:= 'Off',
							sActiveText			:= 'On'
						);

		// Intention:	Set non-concatenated description and objectname with auto-indexing.
		Agg5			: FB_BA_View := (
							iParent				:= THIS^,
							sObjectName	 		:= '{PUM{Idx=5}}',
							sDescription		:= '!{Pump description no concat}'
						);
			Agg5Obj1	: FB_BA_BV_OP := (
							iParent				:= Agg5,
							sObjectName	 		:= '{DST}',
							sDescription		:= '!{Disturbance description no concat}',
							sInactiveText		:= 'Normal',
							sActiveText			:= 'Disturbance'
						);
			Agg5Obj2	: FB_BA_BV_OP := (
							iParent				:= Agg5,
							sObjectName	 		:= '{OPM{Idx=99}}',
							sDescription		:= '{Operation message}',
							sInactiveText		:= 'Off',
							sActiveText			:= 'On'
						);

		// Intention:	Userdefined text wihtout index.
		Agg6			: FB_BA_View := (
							iParent				:= THIS^,
							sObjectName	 		:= '{123A1{!Idx}}',
							sDescription		:= '!{Pump with userdefined label from EPLAN}'
						);
			Agg6Obj1	: FB_BA_BV_OP := (
							iParent				:= Agg6,
							sObjectName	 		:= '{123F1{!Idx}}',
							sDescription		:= '!{Disturbance with userdefined label from EPLAN}',
							sInactiveText		:= 'Normal',
							sActiveText			:= 'Disturbance'
						);
			Agg6Obj2	: FB_BA_BV_OP := (
							iParent				:= Agg6,
							sObjectName	 		:= '{123K1{!Idx}}',
							sDescription		:= '{Operation message with userdefined label from EPLAN}',
							sInactiveText		:= 'Off',
							sActiveText			:= 'On'
						);

		// Intention:	Userdefined, non-concatenated text at aggregate level.
		Agg7			: FB_BA_View := (
							iParent				:= THIS^,
							sObjectName	 		:= '123M1',
							sDescription		:= '!{Pump description non-concatenated}'
						);
			Agg7Obj1	: FB_BA_BV_OP := (
							iParent				:= Agg7,
							sObjectName	 		:= '{DST}',
							sDescription		:= '!{Disturbance description non-concatenated}',
							sInactiveText		:= 'Normal',
							sActiveText			:= 'Disturbance'
						);
			Agg7Obj2	: FB_BA_BV_OP := (
							iParent				:= Agg7,
							sObjectName	 		:= '{OPM{Idx=99}}',
							sDescription		:= '{Operation message}',
							sInactiveText		:= 'Off',
							sActiveText			:= 'On'
						);

		// Intention:	Show an objects instance ID.
		Agg8			: FB_BA_View := (
							iParent				:= THIS^,
							sObjectName	 		:= '{PUM}-ID:{InstID}',
							sDescription		:= '{Pump}-ID:{InstID}'
						);
			Agg8Obj1	: FB_BA_BV_OP := (
							iParent				:= Agg8,
							sObjectName	 		:= '{DST}-ID:{InstID}',
							sDescription		:= '{Disturbance}-ID:{InstID}',
							sInactiveText		:= 'Normal',
							sActiveText			:= 'Disturbance'
						);
			Agg8Obj2	: FB_BA_BV_OP := (
							iParent				:= Agg8,
							sObjectName	 		:= '{OPM}-ID:{InstID}',
							sDescription		:= '{Operation message}-ID:{InstID}',
							sInactiveText		:= 'Off',
							sActiveText			:= 'On'
						);

		// Intention:	Userdefined text wihtout index and non-concatenated objectname (parent-aggregate only).
		Agg9			: FB_BA_View := (
							iParent				:= THIS^,
							sObjectName	 		:= '{223A1{!Idx}}',
							sDescription		:= '!{Pump with userdefined label from EPLAN}',
							eDPADMode			:= E_BA_DPADMode.eIncludeDescription
						);
			Agg9Obj1	: FB_BA_BV_OP := (
							iParent				:= Agg9,
							sObjectName	 		:= '{223F1{!Idx}}',
							sDescription		:= '!{Disturbance with userdefined label from EPLAN}',
							sInactiveText		:= 'Normal',
							sActiveText			:= 'Disturbance'
						);
			Agg9Obj2	: FB_BA_BV_OP := (
							iParent				:= Agg9,
							sObjectName	 		:= '{223K1{!Idx}}',
							sDescription		:= '{Operation message with userdefined label from EPLAN}',
							sInactiveText		:= 'Off',
							sActiveText			:= 'On'
						);
	{endregion}
END_VAR

SUPER^();

//	Default init with auto indexing
Agg1();

Agg1Obj1();
Agg1Obj2();

//	transfer indexinformation into description
Agg2();

Agg2Obj1();
Agg2Obj2();

//	Set objectname and description without labels with auto indexing
Agg3();

Agg3Obj1();
Agg3Obj2();

//	Set objectname and description without labels without auto indexing
Agg4();

Agg4Obj1();
Agg4Obj2();

//	Set description with no concatination and objectname with auto indexing
Agg5();

Agg5Obj1();
Agg5Obj2();

//	Set description with no concatination and objectname with auto indexing
Agg6();

Agg6Obj1();
Agg6Obj2();

//	Userdefined text no concat on aggregate level
Agg7();

Agg7Obj1();
Agg7Obj2();

//	Using attribute so show instance ID
Agg8();

Agg8Obj1();
Agg8Obj2();

//	DPAD mode include description
Agg9();

Agg9Obj1();
Agg9Obj2();

END_FUNCTION_BLOCK

// ---- SAMPLES/Templates/Standard/POUs/Trade/General/EventClasses/FB_BA_EC01.TcPOU
// Template of event classes.
FUNCTION_BLOCK FB_BA_EC01 EXTENDS FB_BA_View
VAR CONSTANT
	OBJECT_NAME			: STRING					:= 'EC{InstID}';
END_VAR
VAR
	{region 'Alarm'}
		AlmSmpl			: FB_BA_EC := (
							iParent					:= THIS^,
							nInstanceID				:= MyECIDs.AlmSmpl,
							sObjectName				:= OBJECT_NAME,
							sDescription			:= '{Alarm (Einfach)}',
							eEventType				:= E_BA_EventType.eAlarm,
							eAlarmMode				:= E_BA_AlarmMode.eSimple,
							aPriority				:= [ 10, 11, 12 ]
						);
		AlmStd			: FB_BA_EC := (
							iParent					:= THIS^,
							nInstanceID				:= MyECIDs.AlmStd,
							sObjectName				:= OBJECT_NAME,
							sDescription			:= '{Alarm (Standard)}',
							eEventType				:= E_BA_EventType.eAlarm,
							eAlarmMode				:= E_BA_AlarmMode.eStandard,
							aPriority				:= [ 13, 14, 15 ]
						);
		AlmExt			: FB_BA_EC := (
							iParent					:= THIS^,
							nInstanceID				:= MyECIDs.AlmExt,
							sObjectName				:= OBJECT_NAME,
							sDescription			:= '{Alarm (Erweitert)}',
							eEventType				:= E_BA_EventType.eAlarm,
							eAlarmMode				:= E_BA_AlarmMode.eExtended,
							aPriority				:= [ 16, 17, 18 ]
						);
	{endregion}
	{region 'Disturb'}
		DstSmpl			: FB_BA_EC	:= (
							iParent					:= THIS^,
							nInstanceID				:= MyECIDs.DstSmpl,
							sObjectName				:= OBJECT_NAME,
							sDescription			:= '{Störung (Einfach)}',
							eEventType				:= E_BA_EventType.eDisturb,
							eAlarmMode				:= E_BA_AlarmMode.eSimple,
							aPriority				:= [ 50, 51, 52 ]
						);
		DstStd			: FB_BA_EC := (
							iParent					:= THIS^,
							nInstanceID				:= MyECIDs.DstStd,
							sObjectName				:= OBJECT_NAME,
							sDescription			:= '{Störung (Standard)}',
							eEventType				:= E_BA_EventType.eDisturb,
							eAlarmMode				:= E_BA_AlarmMode.eStandard,
							aPriority				:= [ 53, 54, 55 ]
						);
		DstExt			: FB_BA_EC := (
							iParent					:= THIS^,
							nInstanceID				:= MyECIDs.DstExt,
							sObjectName				:= OBJECT_NAME,
							sDescription			:= '{Störung (Erweitert)}',
							eEventType				:= E_BA_EventType.eDisturb,
							eAlarmMode				:= E_BA_AlarmMode.eExtended,
							aPriority				:= [ 56, 57, 58 ]
						);
	{endregion}
	{region 'Maintenance'}
		MntnSmpl		: FB_BA_EC := (
							iParent					:= THIS^,
							nInstanceID				:= MyECIDs.MntnSmpl,
							sObjectName				:= OBJECT_NAME,
							sDescription			:= '{Wartung (Einfach)}',
							eEventType				:= E_BA_EventType.eMaintenance,
							eAlarmMode				:= E_BA_AlarmMode.eSimple,
							aPriority				:= [ 90, 91, 92 ]
						);
		MntnStd			: FB_BA_EC := (
							iParent					:= THIS^,
							nInstanceID				:= MyECIDs.MntnStd,
							sObjectName				:= OBJECT_NAME,
							sDescription			:= '{Wartung (Standard)}',
							eEventType				:= E_BA_EventType.eMaintenance,
							eAlarmMode				:= E_BA_AlarmMode.eStandard,
							aPriority				:= [ 93, 94, 95 ]
						);

		MntnExt			: FB_BA_EC := (
							iParent					:= THIS^,
							nInstanceID				:= MyECIDs.MntnExt,
							sObjectName				:= OBJECT_NAME,
							sDescription			:= '{Wartung (Erweitert)}',
							eEventType				:= E_BA_EventType.eMaintenance,
							eAlarmMode				:= E_BA_AlarmMode.eExtended,
							aPriority				:= [ 96, 97, 98 ]
						);
	{endregion}
	{region 'Notification'}
		NtfSmpl			: FB_BA_EC := (
							iParent					:= THIS^,
							nInstanceID				:= MyECIDs.NtfSmpl,
							sObjectName				:= OBJECT_NAME,
							sDescription			:= '{Benachrichtigung (Einfach)}',
							eEventType				:= E_BA_EventType.eNotification,
							eAlarmMode				:= E_BA_AlarmMode.eSimple,
							aPriority				:= [ 130, 131, 132 ]
						);
		NtfStd			: FB_BA_EC := (
							iParent					:= THIS^,
							nInstanceID				:= MyECIDs.NtfStd,
							sObjectName				:= OBJECT_NAME,
							sDescription			:= '{Benachrichtigung (Standard)}',
							eEventType				:= E_BA_EventType.eNotification,
							eAlarmMode				:= E_BA_AlarmMode.eStandard,
							aPriority				:= [ 133, 134, 135 ]
						);
	{endregion}
	{region 'Other'}
		OthSmpl			: FB_BA_EC := (
							iParent					:= THIS^,
							nInstanceID				:= MyECIDs.OthSmpl,
							sObjectName				:= OBJECT_NAME,
							sDescription			:= '{Sonstiges (Einfach)}',
							eEventType				:= E_BA_EventType.eOther,
							eAlarmMode				:= E_BA_AlarmMode.eSimple,
							aPriority				:= [ 180, 181, 182 ]
						);
		OthStd			: FB_BA_EC := (
							iParent					:= THIS^,
							nInstanceID				:= MyECIDs.OthStd,
							sObjectName				:= OBJECT_NAME,
							sDescription			:= '{Sonstiges (Standard)}',
							eEventType				:= E_BA_EventType.eOther,
							eAlarmMode				:= E_BA_AlarmMode.eStandard,
							aPriority				:= [ 183, 184, 185 ]
						);
	{endregion}
END_VAR

SUPER^(); // FB_BA_View
AlmSmpl(); // FB_BA_EC
AlmStd(); // FB_BA_EC
AlmExt(); // FB_BA_EC
DstSmpl(); // FB_BA_EC
DstStd(); // FB_BA_EC
DstExt(); // FB_BA_EC
MntnSmpl(); // FB_BA_EC
MntnStd(); // FB_BA_EC
MntnExt(); // FB_BA_EC
NtfSmpl(); // FB_BA_EC
NtfStd(); // FB_BA_EC
OthSmpl(); // FB_BA_EC
OthStd(); // FB_BA_EC

END_FUNCTION_BLOCK

// ---- SAMPLES/Demo/Objects/Misc/FB_UDef_SpValEx.TcPOU
// User defined setpoint providing value.
// > Contains additional parameters.
FUNCTION_BLOCK FB_UDef_SpValEx EXTENDS FB_UDef_SpVal
VAR_INPUT CONSTANT
	{region 'Variable Parameters'}
		{attribute 'BaParam.Title.DE' := 'Freigabe'}
		{attribute 'BaParam.Title.EN' := 'Enable'}
		{attribute 'BaParam.Access.Read' := 'Guest'}
		{attribute 'BaParam.Access.Write' := 'Advanced'}
		bEnable : BOOL := TRUE;
	{endregion}
END_VAR

SUPER^();

IF (NOT bEnable) THEN
	fResult := 0;
END_IF

END_FUNCTION_BLOCK

// ---- SAMPLES/Demo/Optional Extensions/Events/FB_MyLocalObjectEvents.TcPOU
FUNCTION_BLOCK FB_MyLocalObjectEvents EXTENDS FB_BA_LocalObjectEventSubscriber

METHOD PRIVATE IsPressure : BOOL
VAR_INPUT
	eUnit		: E_BA_Unit;
END_VAR
IsPressure := (E_BA_Unit.ePressure_Pascals <= eUnit) AND_THEN (eUnit <= E_BA_Unit.ePressure_InchesOfMercury);
END_METHOD

METHOD PRIVATE IsTemperature : BOOL
VAR_INPUT
	eUnit		: E_BA_Unit;
END_VAR
IsTemperature := (E_BA_Unit.eTemperature_DegreesCelsius <= eUnit) AND_THEN (eUnit <= E_BA_Unit.eTemperature_DegreeDaysFahrenheit);
END_METHOD

METHOD PROTECTED OnInitInstanceId
VAR_INPUT
	iObject			: I_BA_Object;
END_VAR
VAR_INST
	_nID_Temp		: UDINT						:= 5000;				// First ID to assign to temperature sensors.
	_nID_Prs		: UDINT						:= 6000;				// First ID to assign to pressure sensors.
	_nID_Gen		: UDINT						:= 7000;				// First ID to assign to all other objects.
END_VAR
VAR
	_iAnalogObj		: I_BA_AnalogObject;
	_nID			: REFERENCE TO UDINT;
END_VAR
// Sample 1) Generate instance ID related to configured units.

IF (iObject.InstanceID <> XBA_Globals.nInstId_Auto) THEN
	; // ID already assigned.
ELSIF (iObject.DataClass <> E_BA_DataClass.eAnalog) THEN
	; // Skip.
ELSIF (NOT __QUERYINTERFACE(iObject, _iAnalogObj)) THEN
	; // Failed to convert interface.
ELSE
	// Determine range of instance IDs:
	IF (IsTemperature(_iAnalogObj.Unit)) THEN
		_nID REF= _nID_Temp;
	ELSIF (IsPressure(_iAnalogObj.Unit)) THEN
		_nID REF= _nID_Prs;
	ELSE
		_nID REF= _nID_Gen;
	END_IF
		
	// Assign instance ID:
	_iAnalogObj.InstanceID := _nID;
	iObject.LogMsg.Show1(ADSLOG_MSGTYPE_HINT, 'OIII21', 'Assigned instance ID %d.', F_UDINT(_nID), FALSE);
	
	_nID := (_nID+1);
END_IF
END_METHOD

END_FUNCTION_BLOCK

// ---- SAMPLES/Demo/Optional Extensions/Events/FB_MyProjectEvents.TcPOU
FUNCTION_BLOCK FB_MyProjectEvents EXTENDS FB_BA_ProjectEventSubscriber

METHOD PROTECTED OnProjectStateChanged
VAR_INPUT
	eState			: E_BA_ProjectState;
END_VAR
// Sample 1) Evaluate project state.
CASE (eState) OF
	E_BA_ProjectState.eFirstOpCycle:
		F_BA_LogMessage(ADSLOG_MSGTYPE_HINT, 'OPSC04', 'Initialization done: project is operational.');
	
	E_BA_ProjectState.Error:
		F_BA_LogMessage(ADSLOG_MSGTYPE_HINT, 'OPSC07', 'Initialization failed!');
	
END_CASE
END_METHOD

END_FUNCTION_BLOCK

// ---- SAMPLES/Demo/Plant/FB_Plt_Init1.TcPOU
// How to initialize plant control with parameter builders.
// [Hint]
// > All reference-variables are implemented to ease monitoring of relevant variables.
FUNCTION_BLOCK FB_Plt_Init1 EXTENDS FB_BA_View
VAR
   	{region 'Aggregates'}
		DmprSu_Open							: REFERENCE TO BOOL							REF= DmprSu.bOpen;
		DmprSu_Val							: REFERENCE TO REAL							REF= DmprSu.fActiveVal;
		DmprSu								: FB_TimerAggregateA						:= (iParent:=THIS^,					iLabel:=MyLabels.DmprSu);
		FanSu_Val							: REFERENCE TO UDINT						REF= FanSu.nActiveVal;
		FanSu								: FB_BA_AggregateM							:= (iParent:=THIS^,					iLabel:=MyLabels.FanSu);
			 
		DmprEx_Open							: REFERENCE TO BOOL							REF= DmprEx.bOpen;
		DmprEx_Val							: REFERENCE TO REAL							REF= DmprEx.fActiveVal;
		DmprEx								: FB_TimerAggregateA						:= (iParent:=THIS^,					iLabel:=MyLabels.DmprEx);
		FanEx_Val							: REFERENCE TO UDINT						REF= FanEx.nActiveVal;
		FanEx								: FB_BA_AggregateM							:= (iParent:=THIS^,					iLabel:=MyLabels.FanEx);
			 
		PreHtr_Proc							: REFERENCE TO BOOL							REF= PreHtr.Process.bActive;
		PreHtr_Val							: REFERENCE TO BOOL							REF= PreHtr.bActiveVal;
		PreHtr								: FB_ProcAggregateB							:= (iParent:=THIS^,					iLabel:=MyLabels.PreHtr,			Process:=(iLabel:=MyLabels.ProcPreRinse));
		Erc_Val								: REFERENCE TO BOOL							REF= Erc.bActiveVal;
		Erc									: FB_BA_AggregateB							:= (iParent:=THIS^,					iLabel:=MyLabels.Erc);
		Col_Val								: REFERENCE TO BOOL							REF= Col.bActiveVal;
		Col									: FB_BA_AggregateB							:= (iParent:=THIS^,					iLabel:=MyLabels.Col);
	{endregion}
	{region 'Plant'} 
		OpMode								: E_OpMod_AC								:= E_OpMod_AC.eOff;
		PlantCtrl_OpSta						: REFERENCE TO BOOL							REF= PlantCtrl.bOpSta;
		PlantCtrl_On						: REFERENCE TO BOOL							REF= PlantCtrl.bOn;
		PlantCtrl_PrVal						: REFERENCE TO UDINT						REF= PlantCtrl.nPresentValue;
		PlantCtrl_Step						: REFERENCE TO STRING						REF= PlantCtrl.sStep;
		PlantCtrl							: FB_BA_PlantCtrl := (
												iParent									:= THIS^,
												iLabel									:= MyLabels.PltCtrl,
												stOperation								:= F_BA_PlantOperationBuilder()
																							.AddAggregate(DmprSu,			FALSE,	FALSE,	 T#0S,	 T#0S)
																							.AddAggregate(DmprEx,			FALSE,	FALSE,	 T#0S,	 T#0S)
																							.AddAggregate(PreHtr,			TRUE,	FALSE,	 T#0S,	 T#0S)
																							.AddAggregate(Erc,				FALSE,	FALSE,	 T#0S,	 T#0S)
																							.AddAggregate(Col,				FALSE,	FALSE,	 T#0S,	 T#0S)
																							.AddAggregate(FanSu,			FALSE,	FALSE,	 T#0S,	T#10S)
																							.AddAggregate(FanEx,			FALSE,	FALSE,	T#10S,	 T#0S)
																							.AddOperationMode(E_OpMod_AC.eDisturb, E_BA_Priority.eCritical, E_BA_AggregateIgnoreFlags.Delay)
																								.Close()
																							.AddOperationMode(E_OpMod_AC.eSmokeExtract, E_BA_Priority.eLifeSafety, E_BA_AggregateIgnoreFlags.All)
																								.SetAggregate(DmprSu,		100)
																								.SetAggregate(DmprEx,		100)
																								.SetAggregate(PreHtr,		E_OpMod_Binary.eOn)
																								.SetAggregate(Erc,			E_OpMod_Binary.eOn)
																								.SetAggregate(Col,			E_OpMod_Binary.eOn)
																								.SetAggregate(FanSu,		E_OpMod_Step2.eStep2)
																								.SetAggregate(FanEx,		E_OpMod_Step2.eStep2)
																								.Close()
		// [Bug]								|											.AddOperationMode(E_OpMod_AC.eOff, E_BA_Priority.eProgram, 0)
		// Too large method chain 				|												.Close()
		// will lead to compiler crash :(		|											.AddOperationMode(E_OpMod_AC.eOn, E_BA_Priority.eProgram, 0)
		// Do not use "PlantOperation" builder	|												.SetAggregate(DmprSu,		100)
		// until released.						|												.SetAggregate(DmprEx,		100)
		//										|												.SetAggregate(PreHtr,		E_OpMod_Binary.eOn)
		//										|												.SetAggregate(Erc,			E_OpMod_Binary.eOn)
		//										|												.SetAggregate(Col,			E_OpMod_Binary.eOn)
		//										|												.SetAggregate(FanSu,		E_OpMod_Step2.eStep1)
		//										|												.SetAggregate(FanEx,		E_OpMod_Step2.eStep1)
		//										|												.Close()
		//										|											.AddOperationMode(E_OpMod_AC.eNightCool, E_BA_Priority.eProgram, 0)
		//										|												.SetAggregate(DmprSu,		100)
		//										|												.SetAggregate(DmprEx,		100)
		//										|												.SetAggregate(FanSu,		E_OpMod_Step2.eStep2)
		//										|												.SetAggregate(FanEx,		E_OpMod_Step2.eStep2)
		//										|												.Close()
																							.Build()
											);
	{endregion}
END_VAR

SUPER^(); // FB_BA_View
DmprSu(); // FB_TimerAggregateA
FanSu(bEnCrit := NOT DmprSu.bOpen, nValCrit := E_OpMod_Step2.eOff); // FB_BA_AggregateM
DmprEx(); // FB_TimerAggregateA
FanEx(bEnCrit := NOT DmprEx.bOpen, nValCrit := E_OpMod_Step2.eOff); // FB_BA_AggregateM
PreHtr(); // FB_ProcAggregateB
Erc(); // FB_BA_AggregateB
Col(); // FB_BA_AggregateB
PlantCtrl(nOpMode := OpMode); // FB_BA_PlantCtrl

END_FUNCTION_BLOCK

// ---- SAMPLES/Demo/Supplements/BACnet/Extensions/Events/FB_BACnet_MyLocalObjectEvents.TcPOU
FUNCTION_BLOCK FB_BACnet_MyLocalObjectEvents EXTENDS FB_BA_LocalObjectEventSubscriber

METHOD PROTECTED OnBACnetObjectStateChanged
VAR_INPUT
	iObject			: I_BA_Object;
	fbBACnetObject	: POINTER TO FB_BACnet_BaseObject;
	tState			: TCOM_STATE;
END_VAR
CASE (tState) OF
	TCOM_STATE.TCOM_STATE_PREOP:
		// Sample 1) Enable specific properties.
		CASE (fbBACnetObject^.ObjectType) OF
			E_BACnetObjType.ObjAnalogInput:
				// Sample 1.1) Enable 'PT1 damp factor' for all analog inputs:
				fbBACnetObject^.EnableProperty(E_BACnetPropIdentifier.PropPt1DampFactor, TRUE);
			
		END_CASE
		
		// Sample 2) Writeprotect specific properties.
		CASE (fbBACnetObject^.ObjectType) OF
			E_BACnetObjType.ObjSchedule:
				// Sample 2.1) Writeprotect 'schedule default' for all schedulers:
				fbBACnetObject^.WriteProtectProperty(E_BACnetPropIdentifier.PropScheduleDefault, TRUE);
			
		END_CASE
		
END_CASE
END_METHOD

METHOD PROTECTED OnInitStateChange
VAR_INPUT
	iObject			: I_BA_Object;
	eState			: E_BA_InitState;
END_VAR
VAR
	
	_fbBACnetObj	: POINTER TO FB_BACnet_BaseObject;
END_VAR
// Sample 1) Evaluate object state.
CASE (eState) OF
	E_BA_InitState.ePostInitSupplement:
		// Object has finished to initialize enabled supplement(s).
	
		// Sample 1.1) Initialize some properties:
		IF (iObject.IsReused) THEN
			; // Skip (Do not overwrite previously restored persisted values here).
		ELSIF (iObject.GetBACnetObject(fbObject=>_fbBACnetObj)) THEN
			CASE (_fbBACnetObj^.ObjectType) OF
				E_BACnetObjType.ObjAnalogInput:
					// Write 'PT1 damp factor' for all analog inputs:
					_fbBACnetObj^.WritePropertyReal(E_BACnetPropIdentifier.PropPt1DampFactor, 0.5);
				
			END_CASE
		END_IF

END_CASE
END_METHOD

END_FUNCTION_BLOCK

// ---- SAMPLES/Templates/User-defined/Objects/FB_UDef_Obj.TcPOU
// Some object that only implements a user defined logic.
FUNCTION_BLOCK FB_UDef_Obj EXTENDS FB_BA_Object
VAR_OUTPUT
	nCounter		: UDINT;
END_VAR

SUPER^();

nCounter := (nCounter + 1);

END_FUNCTION_BLOCK
